FUNCTION BuildStringInline : REFERENCE TO StringBuilder255
VAR_INPUT
	value : T_MaxString;
END_VAR
VAR_STAT
	builder : StringBuilder255;
END_VAR

builder.Clear();

builder.Append(value);

BuildStringInline REF= builder;

END_FUNCTION

(* stored: Version 1.1.0.1
   POU BuildStringInline: Id {4bb7c327-72de-4bac-bd0a-0c4baff7eb29}, SpecialFunc None *)
